{attribute 'to_string'}
TYPE E_TableManager_States : (
	TABLEMANAGER_DISABLED
	, TABLEMANAGER_ENABLING
		
	, TABLEMANAGER_INLINE_JOGGING
	, TABLEMANAGER_CROSS_JOGGING
	, TABLEMANAGER_TO_FENCE_JOGGING
	
	, TABLEMANAGER_ROTATE
	, TABLEMANAGER_SELF_CENTER
	
	, TABLEMANAGER_AUTOFEED_OFF
	, TABLEMANAGER_AUTOFEED_ON
	
	, TABLEMANAGER_DOOR_TRACKER_START
	, TABLEMANAGER_DOOR_TRACKER_WAIT_FOR_DATA_READY_OR_TRANSFERRED_IN
	
	, TABLEMANAGER_DOOR_TRACKER_TRANSFERRING_IN
	, TABLEMANAGER_DOOR_TRACKER_ROUTE_READY_WAIT_FOR_FEED_IN
	, TABLEMANAGER_DOOR_TRACKER_DOOR_FEEDING_IN
	, TABLEMANAGER_DOOR_TRACKER_DOOR_IN_MACHINE_IDLE
	, TABLEMANAGER_DOOR_TRACKER_WAIT_FOR_FEED_OUT
	, TABLEMANAGER_DOOR_TRACKER_DOOR_FEEDING_OUT
	, TABLEMANAGER_DOOR_TRACKER_WAIT_ALL_TABLES_READY
	, TABLEMANAGER_DOOR_TRACKER_TRANSFERRING_OUT
	, TABLEMANAGER_DOOR_TRACKER_COMPLETE
	
	, TABLEMANAGER_DOOR_TRACKER_FINDPATH_INIT
	, TABLEMANAGER_DOOR_TRACKER_FINDPATH_RESET
	, TABLEMANAGER_DOOR_TRACKER_FINDPATH_FIND_ENABLED_FEEDOUT_PORTS
	, TABLEMANAGER_DOOR_TRACKER_FINDPATH_WAITING_FOR_CLEAR_ROUTE
	, TABLEMANAGER_DOOR_TRACKER_FINDPATH_FIND_CANDIDATE_ROUTES
	, TABLEMANAGER_DOOR_TRACKER_FINDPATH_FIND_SEARCH_RESULTS
	, TABLEMANAGER_DOOR_TRACKER_FINDPATH_COMPUTE_FINAL_SCORE
	, TABLEMANAGER_DOOR_TRACKER_FINDPATH_REQUEST_NEW_ROUTE_COMPLETE
	, TABLEMANAGER_DOOR_TRACKER_FINDPATH_COMPLETE
	
	, TABLEMANAGER_DOOR_TRACKER_ALL_TARGET_FEEDOUT_PORTS_DISABLED
	, TABLEMANAGER_DOOR_TRACKER_DOOR_HAS_NO_TARGET
	, TABLEMANAGER_ERROR
	
);
END_TYPE

(* stored: Version 1.1.0.1, ProductVersion 3.1.4024.12
   DUT E_TableManager_States: Id {184d05da-20a6-46ec-b011-af3b1f6d5596} *)
